FUNCTION_BLOCK FB_TIIAlarmDbStn
VAR_INPUT
	vIO : ST_DebugStation_VIO;
	NoOfTIIAlm : INT:=NO_OF_TII_SENSOR;
	iLevel : INT:=1;
END_VAR
VAR_OUTPUT
	isTIIError:BOOL;
END_VAR
VAR
	DIFU:R_TRIG;
	tim :TON;
	delay : FB_Delay;
	tPOn: BOOL;	//testerPowerOutoutOn after Delay
	dPOn: BOOL; //dpsPwrbit after Delay
	bitNo:INT;
	almRset:BOOL;
	
	ArrAlmBitBefDelay : ARRAY[1..NO_OF_TII_SENSOR] OF BOOL;
	ArrAlmBitAftDelay : ARRAY[1..NO_OF_TII_SENSOR] OF BOOL;
	ArrAlarmKeepBit	:	ARRAY[1..NO_OF_TII_SENSOR] OF BOOL;
	ArrDelayAlarm : 	ARRAY[1..NO_OF_TII_SENSOR] OF FB_AlarmDelay;
	Arr_ms :			ARRAY[1..NO_OF_TII_SENSOR] OF INT;
	bTIIByPassArray:ARRAY[1..NO_OF_TII_SENSOR] OF BOOL;
	i:INT;
	bTest :BOOL;
END_VAR
VAR_IN_OUT
	
	//bLibError : BOOL;
	//stAlmSubMod:ST_AlarmSubmodules;
	//stAlmMod:ST_AlarmModules;
END_VAR

//<HMI_TII_Test>

	IF bHMITIIBypass THEN
		bTIIByPassArray:= stHMITIIByPassArray[iLevel].bHMITIIByPassArray;
		//FOR i:=1 TO NoOfTIIAlm DO
		//	bTIIByPassArray[i]:= NOT stHMITIIByPassArray[iLevel].bHMITIIByPassArray[i];
		//END_FOR
	ELSE
		FOR i:=1 TO NoOfTIIAlm DO
			//bTIIByPassArray[i]:=bEnableTIIAlarm;
			bTIIByPassArray[i]:=TC_ModuleState[iLevel].TCSite[1].TIERII = E_State.eEnabled;
		END_FOR
	END_IF
//</HMI_TII_Test>
//IF bTest THEN
AlarmUpdate(bENs:=bTIIByPassArray);
//END_IF

METHOD AlarmUpdate : BOOL
VAR
	i						: INT;
	j						: INT;
	_bError					: BOOL;
	iSysAlarmID 			: INT;
	e						: E_TIIAlarm;
	bTstOnCmd 				: BOOL;
	bChkTstOn 				: BOOL;
	
	bAPOnCmd				: BOOL;
	bChkAPOn 				: BOOL;
	//Condition
	lRt:BOOL;
	lEt:BOOL;;
END_VAR

VAR_INPUT
	bENs :ARRAY[1..NO_OF_TII_SENSOR] OF BOOL;
END_VAR

VAR_IN_OUT
	//ArrAlarmKeepBit:ST_AlarmTags;
END_VAR
VAR_OUTPUT
END_VAR
IF iLevel=0 THEN
	RETURN;
END_IF

DIFU(CLK:=vIO.ipDBStnAPPowerOn);
tim(IN:=TRUE,PT:=INT_TO_TIME(1000));
tPOn :=	VIO.bTstDelInt;   //Delay and TesterPwrOnOutput
delay(msec:=100,in:=tPOn,out:=dPOn);

lRt:= FALSE; //:=AP_Deactuated(if AP Down Can Retract)
lEt:= FALSE;

//bTstOnCmd:=vIO.bDPSPowerOnOff;
//bChkTstOn:=vIO.bChkTesterOn;
bAPOnCmd:=vIO.bAP240ACPowerOnOff;
bChkAPOn:=vIO.bChkAP240On;

//<A_Alm_Rst For Door Open TII Alarm>
	IF ALMTC.Level[iLevel].AlarmID[E_TIIAlarm.ipAPPresentSensor] AND vIO.ipDBStnAPPresentSensor THEN
		ALMTC.Level[iLevel].AlarmID[E_TIIAlarm.ipAPPresentSensor] :=FALSE;
	END_IF
//</A_Alm_Rst For Door Open TII Alarm>

FOR i:=1 TO NoOfTIIAlm DO	
	CASE i OF
		E_TIIAlarm.ipAPPresentSensor	   	: e:=E_TIIAlarm.ipAPPresentSensor	   ; ArrAlmBitBefDelay[E_TIIAlarm.ipAPPresentSensor	   	   ]:=	NOT	vIO.ipDBStnAPPresentSensor	  				AND bENs[ 1] ; Arr_ms[e] := 500;  //TIIAlmText[e]:='AP_PresentSensor'  	;//****stTCVIO.iAlarmCode=  E_Alarm.ipAP_PresentSensor 	 ;
        E_TIIAlarm.ipAPPowerOn	 		    : e:=E_TIIAlarm.ipAPPowerOn 		   ; ArrAlmBitBefDelay[E_TIIAlarm.ipAPPowerOn 		   	   ]:=	NOT	vIO.ipDBStnAPPowerOn 	AND bChkAPOn 		AND bENs[ 2] ; Arr_ms[e] := 500;  //TIIAlmText[e]:='AP_PowerOn'	    	; 
	    E_TIIAlarm.ipAPReady				: e:=E_TIIAlarm.ipAPReady		       ; ArrAlmBitBefDelay[E_TIIAlarm.ipAPReady		       	   ]:=	NOT	vIO.ipDBStnAPReady	AND vIO.ipDBStnAPPresentSensor	AND bENs[ 3] ; Arr_ms[e] := 500;  //TIIAlmText[e]:='AP_Ready' 		    	;      
	    //E_TIIAlarm.ipAPDeactuatedPLC		: e:=E_TIIAlarm.ipAPDeactuatedPLC	   ; ArrAlmBitBefDelay[E_TIIAlarm.ipAPDeactuatedPLC	   	   ]:=	NOT	vIO.ipDBStnHandlerSafeToEnterPLC	  				AND bENs[ 4] ; Arr_ms[e] := 500;  (*TIIAlmText[e]:='AP_DeactuatedPLC' 		*);   
	    //E_TIIAlarm.ipAPDeactuatedHwr		: e:=E_TIIAlarm.ipAPDeactuatedHwr	   ; ArrAlmBitBefDelay[E_TIIAlarm.ipAPDeactuatedHwr	   	   ]:=	NOT	vIO.ipDBStnHandlerSafeToEnterHwr	  				AND bENs[ 5] ; Arr_ms[e] := 500;  (*TIIAlmText[e]:='AP_DeactuatedHwr' 		*); 
//	    E_TIIAlarm.ipCellFluidLeakage1		: e:=E_TIIAlarm.ipCellFluidLeakage1	   ; ArrAlmBitBefDelay[E_TIIAlarm.ipCellFluidLeakage1	   ]:=	vIO.ipCellFluidLeakage1	  					AND bENs[ 6] ; Arr_ms[e] := 500;  (*TIIAlmText[e]:='CellFluidLeakage1' 	*);   
//	    E_TIIAlarm.ipCellFluidLeakage2		: e:=E_TIIAlarm.ipCellFluidLeakage2	   ; ArrAlmBitBefDelay[E_TIIAlarm.ipCellFluidLeakage2	   ]:=	vIO.ipCellFluidLeakage2	  					AND bENs[ 7] ; Arr_ms[e] := 500;  (*TIIAlmText[e]:='CellFluidLeakage2' 	*);   
	    E_TIIAlarm.ipCellGroundFault 		: e:=E_TIIAlarm.ipCellGroundFault 	   ; ArrAlmBitBefDelay[E_TIIAlarm.ipCellGroundFault 	   ]:=		vIO.ipDBStnCellGroundFault 	  				AND bENs[ 8] ; Arr_ms[e] := 500;  //TIIAlmText[e]:='CellGroundFault'  		;
//        E_TIIAlarm.ipTesterPresent			: e:=E_TIIAlarm.ipTesterPresent	       ; ArrAlmBitBefDelay[E_TIIAlarm.ipTesterPresent	       ]:=	NOT	vIO.ipTesterPresent	 AND bTstOnCmd 		AND bENs[ 9] ; Arr_ms[e] := 500;  (*TIIAlmText[e]:='TesterPresent' 		*);
//        E_TIIAlarm.ipTesterPowerOn			: e:=E_TIIAlarm.ipTesterPowerOn	       ; ArrAlmBitBefDelay[E_TIIAlarm.ipTesterPowerOn	       ]:=	NOT	vIO.ipTesterPowerOn  	AND bChkTstOn 	AND bENs[10] ; Arr_ms[e] := 500;  (*TIIAlmText[e]:='TesterPowerOn' 		*);    
//        E_TIIAlarm.ipTesterReady			: e:=E_TIIAlarm.ipTesterReady	       ; ArrAlmBitBefDelay[E_TIIAlarm.ipTesterReady	           ]:=	NOT	vIO.ipTesterReady	     	 			AND bENs[11] ; Arr_ms[e] := 500;  (*TIIAlmText[e]:='TesterReady'       	*);   
//       	E_TIIAlarm.ipTCCellDoorClosed		: e:=E_TIIAlarm.ipTCCellDoorClosed	   ; ArrAlmBitBefDelay[E_TIIAlarm.ipTCCellDoorClosed	   ]:=	NOT	vIO.ipTCCellDoorClosed	  				AND bENs[12] ; Arr_ms[e] := 500;  (*TIIAlmText[e]:='TCCellDoorClosed' 		*);
//        E_TIIAlarm.ipTesterLatchesClosed	: e:=E_TIIAlarm.ipTesterLatchesClosed  ; ArrAlmBitBefDelay[E_TIIAlarm.ipTesterLatchesClosed    ]:=	NOT	vIO.ipTesterLatchesClosed AND bTstOnCmd AND bENs[13] ; Arr_ms[e] := 500;  (*TIIAlmText[e]:='TesterLatchesClosed' 	*);
//        E_TIIAlarm.ipTIUPresent			    : e:=E_TIIAlarm.ipTIUPresent	       ; ArrAlmBitBefDelay[E_TIIAlarm.ipTIUPresent	           ]:=	NOT	vIO.ipTIUPresent	      				AND bENs[14] ; Arr_ms[e] := 500;  (*TIIAlmText[e]:='TIUPresent' 	      	*);
//        E_TIIAlarm.ipTCDrawerCylExtendRS	: e:=E_TIIAlarm.ipTCDrawerCylExtendRS  ; ArrAlmBitBefDelay[E_TIIAlarm.ipTCDrawerCylExtendRS    ]:=		vIO.ipTCDrawerCylExtendRS	AND lEt		AND bENs[15] ; Arr_ms[e] := 500;  (*TIIAlmText[e]:='TCDrawerCylExtendRS' 	*);
//        E_TIIAlarm.ipTCDrawerCylRetractRS	: e:=E_TIIAlarm.ipTCDrawerCylRetractRS ; ArrAlmBitBefDelay[E_TIIAlarm.ipTCDrawerCylRetractRS   ]:=		vIO.ipTCDrawerCylRetractRS	AND	lRt		AND bENs[16] ; Arr_ms[e] := 500;  (*TIIAlmText[e]:='TCDrawerCylRetractRS'	*);
                   
                   
	               
		//E_Alarm.LibraryCylErr			:	ArrAlmBitBefDelay[E_Alarm.LibraryCylErr				]:=bError(*From Lib*) AND E_Alarm.LibraryCylErr == LibErrorID  ; ArrMiliSecond[E_Alarm.LibraryCylErr   ] := 0;		
	
	END_CASE

	//Delay Library Alm Bit
	ArrDelayAlarm[i](	alarmState			:= ArrAlmBitBefDelay[i],
						triggerAlarmState	=> ArrAlmBitAftDelay[i],
						msec				:= Arr_ms[i]);	//DelayAlmBit
	

	IF ArrAlmBitAftDelay[i] THEN					//realtime IO update array
		//stAlmMod.Level[iLevel].AlarmID[i]:=TRUE;
		ALMTC.Level[iLevel].AlarmID[i]:=TRUE;
	ELSE
		//TIIAlmText[i]:='';  
	END_IF		
		//_bError := _bError OR stAlmMod.Level[iLevel].AlarmID[i];
		_bError := _bError OR ALMTC.Level[iLevel].AlarmID[i];
	
END_FOR
isTIIError := _bError ;  //bError refers to system Error;

(*
//Alarm Reset ===========================================================================
IF almRset THEN
	IF ArrAlmSubModule.AlarmSubmodule[iSubMod].ArrAlarmKeepBit[bitNo] THEN
		ArrAlmSubModule.AlarmSubmodule[iSubMod].ArrAlarmKeepBit[bitNo] := FALSE;
	END_IF
END_IF
//=======================================================================================
*)
END_METHOD

END_FUNCTION_BLOCK

(* stored: Version 1.1.0.1, ProductVersion 3.1.4022.18
   POU FB_TIIAlarmDbStn: Id {1f1c0a9a-a15d-4901-bcd2-0649d00aa61a}, SpecialFunc None
   Method AlarmUpdate: Id {df4f023a-29b0-4ee7-baee-77dc81ad8f78} *)
